FUNCTION_BLOCK System_TaskInfo
VAR_INPUT
	
END_VAR
VAR_OUTPUT
	// Object ID of the task reference, from which the PLC program is called.
	ObjId: UDINT;
	// Set task cycle time in multiples of 100 ns
	CycleTime: UDINT;
	// Set task priority
	Priority: UINT;
	// ADS port of the task
	AdsPort: UINT;
	(* 
	Cycle counter
	Please note that the cycle counter refers to the actual system task 
	and not to the task reference of the PLC project. The background to 
	this is that several PLC projects or other TcCOM modules can share 
	a task and these modules can thus access the same cycle counter. 
	As a result, the cycle counter is reset during a TwinCAT restart in 
	RUN mode (and not when resetting the PLC project). *)
	CycleCount: UDINT;
	// Distributed Clock System Time. It remains constant for a task runtime.
	DcTaskTime: LINT;
	// Cycle time required for the last cycle in multiples of 100 ns
	LastExecTime: UDINT;
	// During the first PLC task cycle, this variable has the value TRUE.
	FirstCycle: BOOL;
	(* 
	This variable indicates whether the set task cycle time was exceeded.
	The value of the CycleTimeExceeded variable is updated in each cycle. 
	The variable is set to 0 if the previous cycle has been completed 
	within its intended timeframe, otherwise to 1. *)
	CycleTimeExceeded: BOOL;
	(* 
	This variable has the value TRUE if the origin of the current call 
	is declared with the attribute 'TcCallAfterOutputUpdate'. *)
	InCallAfterOutputUpdate: BOOL;
	(* This variable has the value TRUE if the real-time limit is 
	exceeded on a mixed core (Windows + real-time on one core). In this 
	case the value TRUE refers to the core on which the corresponding 
	task is running. *)
	RTViolation: BOOL;
	// Name of the task reference object in the PLC project (e.g. 'MyPlcProject_PlcTaskRef')
	TaskName: STRING(63);
END_VAR
VAR
	
	_ThisTaskInfo: PlcTaskSystemInfo;
	_AllTaskInfo : ARRAY[0..10] OF PlcTaskSystemInfo;
	index : UDINT;
	TaskCount : UDINT;
	TaskIndex : DINT ;
	
	
END_VAR

TaskCount := TwinCAT_SystemInfoVarList._AppInfo.TaskCnt;
FOR index := 1 TO LIMIT(1,TaskCount,10)  DO
	_AllTaskInfo[index] := TwinCAT_SystemInfoVarList._TaskInfo[index];
END_FOR
TaskIndex := GETCURTASKINDEXEX();
_ThisTaskInfo := _AllTaskInfo[TaskIndex];

_ThisTaskInfo := _TaskInfo[TaskIndex];
ObjId := _ThisTaskInfo.ObjId; 
CycleTime := _ThisTaskInfo.CycleTime;
Priority := _ThisTaskInfo.Priority;
AdsPort := _ThisTaskInfo.AdsPort;
CycleCount := _ThisTaskInfo.CycleCount;
DcTaskTime := _ThisTaskInfo.DcTaskTime;
LastExecTime := _ThisTaskInfo.LastExecTime;
FirstCycle := _ThisTaskInfo.FirstCycle;
CycleTimeExceeded := _ThisTaskInfo.CycleTimeExceeded;
InCallAfterOutputUpdate := _ThisTaskInfo.InCallAfterOutputUpdate;
RTViolation := _ThisTaskInfo.RTViolation;

TaskName := _ThisTaskInfo.TaskName;

METHOD getCurrentTaskInfo : REFERENCE TO PlcTaskSystemInfo
VAR_INPUT
END_VAR
getCurrentTaskInfo REF= _ThisTaskInfo;
END_METHOD

METHOD getTaskCount : UDINT
VAR_INPUT
END_VAR
getTaskCount := _AppInfo.TaskCnt;
END_METHOD

METHOD getTaskFirstIndex : UDINT
VAR_INPUT
END_VAR
getTaskFirstIndex := 1;
END_METHOD

METHOD getTaskInfoByIndex : REFERENCE TO PlcTaskSystemInfo
VAR_INPUT
	Index : UDINT;
END_VAR
IF Index >= 1 AND index <= 10 THEN
	getTaskInfoByIndex REF= _AllTaskInfo[Index];
ELSE
	getTaskInfoByIndex REF= _AllTaskInfo[0];
END_IF
END_METHOD

END_FUNCTION_BLOCK

(* stored: Version 1.1.0.1, ProductVersion 3.1.4024.12
   POU System_TaskInfo: Id {23e4a9df-9958-46d3-9111-ab3ad0dae806}, SpecialFunc None
   Method getCurrentTaskInfo: Id {eabed3e6-3b9b-466c-9829-15399749e77c}
   Method getTaskCount: Id {b0ba8701-2c67-4361-80c2-81c8bddbc1ba}
   Method getTaskFirstIndex: Id {498d1279-57c5-48ef-8a5b-4dab9231d9d5}
   Method getTaskInfoByIndex: Id {1b42230b-8a39-4361-8e6b-25071b433320} *)
